(* CoDeSys 2.3.9.48 project: Only485.pro *)
(* Libraries: C:\Program Files (x86)\3S Software\CODESYS V2.3\Targets\WAGO\Libraries\Serial_Interface_01.lib 25.1.13 07:35:32, SerComm.lib 31.5.11 09:06:48, Standard.lib 8.11.10 12:37:48, SYSLIBCALLBACK.LIB 8.11.10 12:37:48 *)

(* PLC configuration (modules and I/O channels)
K-Bus [K_Bus] node 0, in %IB0 out %QB0
  0750-0652#24 RS-232/RS-485 Interface adjustable (24 Bytes) [Type_30_1_Channels] node 0, in %IB28 out %QB28 {INTTypePAAssignment = PLC; INTTypeModule = plugged}
    AT %IB0 [BYTEOnB_I] First Byte of 24
    AT %QB0 [BYTEOnB_Q] First Byte of 24
  0750-0653/0003-0000#03 RS485 Interface (Adjustable), 3 Bytes [Type_21_1_Channels] node 0, in %IB28 out %QB28 {INTTypePAAssignment = PLC; INTTypeModule = plugged}
    AT %IX12.0 [BOOLOnX_I] Transmission acknowledgement
    AT %IX12.1 [BOOLOnX_I] Reception request
    AT %IX12.2 [BOOLOnX_I] Initialization acknowledgement
    AT %IX12.3 [BOOLOnX_I] Input buffer is full
    AT %IX12.4 [BOOLOnX_I] Number of received characters Bit 0
    AT %IX12.5 [BOOLOnX_I] Number of received characters Bit 1
    AT %IX12.6 [BOOLOnX_I] Number of received characters Bit 2
    AT %IB25 [BYTEOnB_I] Input data Byte 0
    AT %IB26 [BYTEOnB_I] Input data Byte 1
    AT %IB27 [BYTEOnB_I] Input data Byte 2
    AT %QX12.0 [BOOLOnX_Q] Transmission request
    AT %QX12.1 [BOOLOnX_Q] Reception acknowledgement
    AT %QX12.2 [BOOLOnX_Q] Initialization request
    AT %QX12.4 [BOOLOnX_Q] Number of characters Bit 0
    AT %QX12.5 [BOOLOnX_Q] Number of characters Bit 1
    AT %QX12.6 [BOOLOnX_Q] Number of characters Bit 2
    AT %QB25 [BYTEOnB_Q] Output data Byte 0
    AT %QB26 [BYTEOnB_Q] Output data Byte 1
    AT %QB27 [BYTEOnB_Q] Output data Byte 2
  0750-0653/0003-0000#03 RS485 Interface (Adjustable), 3 Bytes [Type_21_1_Channels] node 0, in %IB52 out %QB52 {INTTypePAAssignment = PLC; INTTypeModule = plugged}
    AT %IX14.0 [BOOLOnX_I] Transmission acknowledgement
    AT %IX14.1 [BOOLOnX_I] Reception request
    AT %IX14.2 [BOOLOnX_I] Initialization acknowledgement
    AT %IX14.3 [BOOLOnX_I] Input buffer is full
    AT %IX14.4 [BOOLOnX_I] Number of received characters Bit 0
    AT %IX14.5 [BOOLOnX_I] Number of received characters Bit 1
    AT %IX14.6 [BOOLOnX_I] Number of received characters Bit 2
    AT %IB29 [BYTEOnB_I] Input data Byte 0
    AT %IB30 [BYTEOnB_I] Input data Byte 1
    AT %IB31 [BYTEOnB_I] Input data Byte 2
    AT %QX14.0 [BOOLOnX_Q] Transmission request
    AT %QX14.1 [BOOLOnX_Q] Reception acknowledgement
    AT %QX14.2 [BOOLOnX_Q] Initialization request
    AT %QX14.4 [BOOLOnX_Q] Number of characters Bit 0
    AT %QX14.5 [BOOLOnX_Q] Number of characters Bit 1
    AT %QX14.6 [BOOLOnX_Q] Number of characters Bit 2
    AT %QB29 [BYTEOnB_Q] Output data Byte 0
    AT %QB30 [BYTEOnB_Q] Output data Byte 1
    AT %QB31 [BYTEOnB_Q] Output data Byte 2
Fieldbus variables [FB_VARS] node 1, in %IB0 out %QB0
Flag variables [FLAG_VARS] node 2, in %IB0 out %QB0
Modbus-Master [MB_MASTER] node 3, in %IB0 out %QB0
*)

(* Task configuration *)
TASK Ser485 (PRIORITY := 1, INTERVAL := T#1500ms);
	PLC_PRG();
END_TASK

(* POU PLC_PRG, ST *)
PROGRAM PLC_PRG
VAR
	 iBytesToSend : INT;
    TimeCycleDiff : TIME;
    TimeSendDiff : TIME;
    iCycleCountDiff:INT;

    i                 : INT;

    TimeAct : TIME;
    TimeSendOld: TIME;
    TimeCycleOld : TIME;

    iCycleCount : INT;
    iCycleCountOld:INT;

    iCount2:INT;
    xInitDone:BOOL := FALSE;

    baSendBuffer:ARRAY [0..99] OF BYTE;



(* COM2  ********************************************)
    COM3             : SERIAL_INTERFACE;
    xOpenPort2        : BOOL := TRUE;
    xInitPort2        : BOOL;
    xSendActive2    : BOOL;
       xSendActive2Old : BOOL;
    SendString2        : STRING(100) := '0123456789012345678901234567890123456789012345678901234567890123456789012345678901234567890123456789';
    (*SendString2        : STRING := '01234567890123456789012345678901234567890123456789012345678901234567890123456789';*)
    (*SendString2        : STRING := '01234567890123456789';*)
    ReceiveBuffer2    : typRing_Buffer;

    ReceiveBuffer2OldIndex    : INT;
    ReceiveString2     : STRING(255);
    pReceiveStr2      : POINTER TO ARRAY[0..255] OF BYTE;
    help2Idx         : INT;
    iTo2            : INT;

END_VAR
TimeAct := TIME();
iCycleCount := iCycleCount+1;

IF (NOT xInitDone) THEN
    iBytesToSend := SIZEOF(baSendBuffer);

    FOR i:=0 TO iBytesToSend DO
        baSendBuffer[i] := INT_TO_BYTE (i);
    END_FOR
    xInitDone := TRUE;
END_IF

(* Send and Receive for COM2 *)
COM3(    bCOM_PORT_NR     := 16#03,
	 xOPEN_COM_PORT     := xOpenPort2,
	cbBAUDRATE         := BAUD_57600,
        cbsBYTESIZE        := BS_8,
        cpPARITY        := PARITY_NO,
        csSTOPBITS        := STOPBITS_1,
        cfFLOW_CONTROL    := HALFDUPLEX,
        (*cfFLOW_CONTROL    := NCS_NO_FLOW_CONTROL,*)
        utRECEIVE_BUFFER := ReceiveBuffer2,
        ptSEND_BUFFER    := ADR(baSendBuffer),
        xINIT            := xInitPort2,
        iBYTES_TO_SEND    := iBytesToSend,
        xSTART_SEND        := xSendActive2 );


IF (COM3.Com_Port_Ist_Offen) THEN

    IF (xSendActive2 AND NOT xSendActive2Old) THEN
        TimeSendOld := TimeAct;
        iCycleCountOld := iCycleCount;
    END_IF
    IF (NOT xSendActive2 AND  xSendActive2Old) THEN
        TimeSendDiff := TimeAct - TimeSendOld;
        iCycleCountDiff := iCycleCount-iCycleCountOld;
    END_IF
    xSendActive2Old := xSendActive2;

    TimeCycleDiff := TimeAct - TimeCycleOld;
    TimeCycleOld := TimeAct;
    IF (NOT xSendActive2) THEN
        iCount2 := (iCount2+1)MOD 100;
        IF (iCount2 =0) THEN
            xSendActive2 := NOT xSendActive2;
        END_IF
    END_IF
END_IF
END_PROGRAM
